FUNCTION_BLOCK FB_Event EXTENDS FB_ListString IMPLEMENTS I_Event
VAR_INPUT
END_VAR
VAR_OUTPUT
END_VAR
VAR
	iParent:			I_Component;
	iLogger:			I_Logger;
	stEvent:			ST_Event;
END_VAR

SUPER^();

METHOD FB_init : BOOL
VAR_INPUT
	bInitRetains : BOOL; // if TRUE, the retain variables are initialized (warm start / cold start)
	bInCopyCode : BOOL;  // if TRUE, the instance afterwards gets moved into the copy code (online change)
	iParent:			I_Component;
END_VAR
THIS^.iParent:= iParent;
END_METHOD

METHOD INTERNAL M_Arguments : STRING(255)
VAR_INPUT
END_VAR
VAR
	nIndex:			INT;
END_VAR
WHILE nIndex < nLength DO
	M_Arguments:= Concat(Concat(M_Arguments, pList[nIndex]), '$N');
	nIndex:= nIndex + 1;
END_WHILE
END_METHOD

METHOD PUBLIC M_Debug : BOOL
VAR_INPUT
	Message:				STRING(255);
END_VAR
END_METHOD

METHOD PUBLIC M_Error : BOOL
VAR_INPUT
	Message:				STRING(255);
	ID:						UDINT;
	Severity:				E_Severity;
END_VAR
stEvent.Source:= iParent;
stEvent.EventType:= E_Event.Error;
stEvent.Timestamp:= F_GetSystemTime();
stEvent.ID:= ID;
stEvent.Message:= Message;
stEvent.Arguments:= M_Arguments();
stEvent.Active:= TRUE;

IF Severity >= E_Severity.Abort THEN
	iParent.M_Request(E_Request.Abort);
ELSIF Severity >= E_Severity.Stop THEN
	iParent.M_Request(E_Request.Stop);
ELSIF Severity >= E_Severity.Complete THEN	
	iParent.M_Request(E_Request.Complete);
ELSIF Severity >= E_Severity.Hold THEN
	iParent.M_Request(E_Request.Hold);
ELSIF Severity >= E_Severity.Pause THEN
	iParent.M_Request(E_Request.Pause);
END_IF

IF iLogger <> 0 THEN
	iLogger.M_Log(stEvent);
END_IF

M_Clear();
END_METHOD

METHOD PUBLIC M_Information : BOOL
VAR_INPUT
	Message:				STRING(255);
	ID:						UDINT;
END_VAR
END_METHOD

METHOD PUBLIC M_Warning : BOOL
VAR_INPUT
	Message:				STRING(255);
	ID:						UDINT;
END_VAR
END_METHOD

PROPERTY PUBLIC P_Logger : I_Logger
GET
P_Logger:= iLogger;
END_GET
SET
iLogger:= P_Logger;
END_SET
END_PROPERTY

END_FUNCTION_BLOCK

(* stored: Version 1.1.0.1
   POU FB_Event: Id {59616103-7f2e-4b6f-81bd-583969a36d28}, SpecialFunc None
   Method FB_init: Id {be23ffcc-529d-4010-ace3-b17baed191a5}
   Method M_Arguments: Id {70779266-7b36-4bce-9e6f-049e951fd75a}
   Method M_Debug: Id {0a2b992b-2a4a-0251-0210-713b326debf6}
   Method M_Error: Id {55348828-4763-4c06-9dd1-090fa29a8379}
   Method M_Information: Id {d9a244f2-1d6f-434f-aab4-cad6aacbb94f}
   Method M_Warning: Id {d443b8bb-774e-487e-80a2-79cf66a0376c}
   Property P_Logger: Id {642d0edf-ded0-4248-be29-8384d3180124}
   Get Get: Id {99e41819-eb78-4b29-b3e9-6728532b14b1}
   Set Set: Id {be31597a-6e88-476b-aec8-980317d6bc1a} *)
